(* PLC project BlogProject.project, CODESYS CODESYS V3.5 SP14 Patch 3 *)
(* stored: creationDateTime 2021-10-07T21:04:37.3452952, modificationDateTime 2021-10-07T20:40:20.1109198 *)

FUNCTION_BLOCK MC_CORE
  VAR_INPUT
    System : POINTER TO udtSystem;
  END_VAR
  VAR
    Stage : INT;  (* Счетчик стадий для цикда *)
    events : BOOL;  (* проверка выполнения всех условий *)
  END_VAR
  VAR CONSTANT
    Max_Stage : INT := 9;  (* Максимальное количество состояний системы *)
  END_VAR

            FOR Stage:=0 TO Max_Stage DO
	IF System^.eCurrentState = System^.arTransactions[Stage].eCurrentState THEN
		events:= System^.arTransactions[Stage].mcEvent_1.getEvent() AND System^.arTransactions[Stage].mcEvent_2.getEvent(); 
		IF events THEN
			System^.arTransactions[Stage].mcAction_1.getAction();
			System^.arTransactions[Stage].mcAction_2.getAction();
			System^.eCurrentState:=System^.arTransactions[Stage].eNextStage;
			EXIT;
		END_IF
	END_IF	
END_FOR
          
END_FUNCTION_BLOCK
